(* CoDeSys 2.3.9.37 project: CapB_2.pro *)
(* Libraries: Standard.lib 4.10.05 12:14:46 *)

(* POU PLC_PRG, ST *)
PROGRAM PLC_PRG
VAR
  Alarma:BOOL;
  posx:INT:=0;
  posy:INT:=0;
  angulo:INT:=0;
  escala:INT:=0;
	subex: BOOL;
	bajax: BOOL;
	subey: BOOL;
	bajay: BOOL;
	subeang: BOOL;
	bajaang: BOOL;
	subeesc: BOOL;
	bajaesc: BOOL;
END_VAR
IF subex THEN
    posx:=posx+1;
END_IF


IF bajax THEN
    posx:=posx-1;
END_IF


IF subey THEN
    posy:=posy+1;
END_IF


IF bajay THEN
    posy:=posy-1;
END_IF



IF subeesc THEN
    escala:=escala+1;
END_IF


IF bajaesc THEN
    escala:=escala-1;
END_IF


IF subeang THEN
    angulo:=angulo+1;
END_IF


IF bajaang THEN
    angulo:=angulo-1;
END_IF
END_PROGRAM

(* Visualisation EjemploVisu
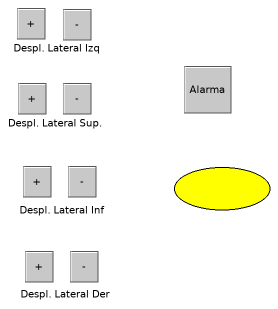
button at (35,35)-(63,66): text "+"; taps PLC_PRG.subex
button at (81,36)-(109,67): text "-"; taps PLC_PRG.bajax
ellipse at (192,194)-(288,237): alarm colour if PLC_PRG.Alarma; left PLC_PRG.posx; top PLC_PRG.posy; right PLC_PRG.escala; bottom PLC_PRG.angulo
button at (36,110)-(64,141): text "+"; taps PLC_PRG.subey
button at (81,110)-(109,141): text "-"; taps PLC_PRG.bajay
button at (41,193)-(69,224): text "+"; taps PLC_PRG.subeang
button at (86,193)-(114,224): text "-"; taps PLC_PRG.bajaang
button at (43,278)-(71,309): text "+"; taps PLC_PRG.subeesc
button at (88,278)-(116,309): text "-"; taps PLC_PRG.bajaesc
rectangle at (6,60)-(144,90): text "Despl. Lateral Izq"
rectangle at (4,135)-(142,165): text "Despl. Lateral Sup."
rectangle at (11,222)-(149,252): text "Despl. Lateral Inf"
rectangle at (14,306)-(152,336): text "Despl. Lateral Der"
button at (202,93)-(249,140): text "Alarma"; toggles PLC_PRG.Alarma
*)
